{attribute 'hide'}
FUNCTION_BLOCK FileEntry_Test EXTENDS TcUnit.FB_TestSuite

IsFileReturnsExpected();
NameReturnsExpected();
GetFullPathReturnsExpected();

METHOD GetFullPathReturnsExpected
VAR
	expected : FileName;
	actual : FileName;
	fileEntry : FileEntry('C:\temp', 'test.txt');
END_VAR
TEST('GetFullPathReturnsExpected');

// @TEST-FIXTURE

// @TEST-RUN
expected := 'C:\temp\test.txt';
actual := fileEntry.GetFullPath();

// @TEST-ASSSERT
AssertEquals_STRING(Expected := expected, Actual := actual, Message := 'File GetFullPath did not return expected');

TEST_FINISHED();
END_METHOD

METHOD IsFileReturnsExpected
VAR
	result : BOOL;
	fileEntry : FileEntry('', '');
END_VAR
TEST('IsFileReturnsExpected');

// @TEST-FIXTURE

// @TEST-RUN
result := fileEntry.IsFile;

// @TEST-ASSSERT
AssertTrue(Condition := result, Message := 'IsFile did not return TRUE');

TEST_FINISHED();
END_METHOD

METHOD NameReturnsExpected
VAR
	expected : FileName;
	actual : FileName;
	fileEntry : FileEntry('C:\temp', 'test.txt');
END_VAR
TEST('NameReturnsExpected');

// @TEST-FIXTURE

// @TEST-RUN
expected := 'test.txt';
actual := fileEntry.Name;

// @TEST-ASSSERT
AssertEquals_STRING(Expected := expected, Actual := actual, Message := 'File name did not return expected');

TEST_FINISHED();
END_METHOD

END_FUNCTION_BLOCK

(* stored: Version 1.1.0.1, ProductVersion 3.1.4024.9
   POU FileEntry_Test: Id {17041bfc-bd21-46d0-83c0-0d4172417c38}, SpecialFunc None
   Method GetFullPathReturnsExpected: Id {41bb275b-6cd0-4836-90c9-4cd1077b2f6d}
   Method IsFileReturnsExpected: Id {3436b61c-0f7a-44b8-8996-82a32d002ec6}
   Method NameReturnsExpected: Id {53e200f9-6afe-4bd6-b22b-6d31a0529872} *)
